(*
SPDX-FileCopyrightText: © 2026 Oleksandr Tiutyk <trofimich@gmail.com>
SPDX-License-Identifier: MIT
License: https://opensource.org/license/mit
*)

(*!
<summary>Enumerates a borrowed collection using an independent cursor.</summary>
<description>
The source must be non-null, outlive the cursor and remain structurally unchanged during traversal. The caller
explicitly releases a dynamically created cursor. Current borrows a byte cached in this cursor, not the source
buffer; it never transfers ownership. MoveNext stops advancing at the end position of an unchanged source;
repeated exhausted calls return FALSE until Reset.
A null constructor source is diagnosed by traversal/current access, never by FB_init.
</description>
*)

{attribute 'no_explicit_call' := 'do not call this function block directly'}
{attribute 'enable_dynamic_creation'}
FUNCTION_BLOCK ByteListEnumerator EXTENDS TOF_Core.Object IMPLEMENTS TOF_Core.IEnumerator
VAR_STAT
	//! <summary>Class name shared by all instances of this function block.</summary>
	{attribute 'hide'} 
	_ClassName : STRING := __POUNAME();
END_VAR
VAR
	{attribute 'hide'} 
	_List : IReadOnlyByteList;
	{attribute 'hide'} 
	_CurrentIndex : DINT := -1;
	
	{attribute 'hide'} 
	_CurrentByte : BYTE;
	{attribute 'hide'} 
	_GenericValue : TOF_Core.GENERIC_VALUE;	
END_VAR

(*!
<summary>Borrows the concrete cursor class name without transferring storage ownership.</summary>
*)
{attribute 'monitoring' := 'call'}
PROPERTY ClassName : REFERENCE TO STRING
GET
ClassName REF= _ClassName;
END_GET
END_PROPERTY

(*!
<summary>Exposes a read-only borrowed view of the current entry.</summary>
<description>
Reading Current before the first successful MoveNext, after Reset or after exhaustion yields an empty
descriptor. At a valid position, the source byte is copied into cursor-local storage and the returned
descriptor borrows that storage, including when the byte value is zero. Do not modify or release the
descriptor. Keep the cursor alive while using the view; subsequent Current access can overwrite its cached
byte. Cursor movement or reset invalidates the previous view contract.
Missing source raises DataMemberNotSpecifiedException before source access or cursor advancement.
</description>
*)
{attribute 'monitoring' := 'call'}
PROPERTY FINAL Current : REFERENCE TO TOF_Core.GENERIC_VALUE
GET
requireSource();

IF _CurrentIndex >= 0 AND_THEN _CurrentIndex < _List.Length THEN
	_CurrentByte := _List.Get(index := _CurrentIndex); 
	_GenericValue := TOF_Core.GenericValueFactory.FromParts(
		genericTypeClass := TOF_Core.GENERIC_TYPE_CLASS.UINT_8,
		address := ADR(_CurrentByte),
		size := 1,
		memoryManagementBehavior := TOF_Core.GENERIC_MEMORY_MANAGEMENT_BEHAVIOR.STORE_ORIGINAL_REFERENCE_AND_NOT_OWNS_MEMORY
	);
ELSE
	_GenericValue.Reset();
END_IF 

Current REF= _GenericValue;
END_GET
END_PROPERTY

(*!
<summary>Returns the current entry in its concrete representation.</summary>
<description>
Use only after MoveNext returns TRUE and before the next cursor or source change. No result is promised
outside a valid position. The byte is returned by value.
Missing source raises DataMemberNotSpecifiedException before source access or cursor advancement.
</description>
*)
{attribute 'monitoring' := 'call'}
PROPERTY FINAL CurrentByte : BYTE
GET
requireSource();

IF _CurrentIndex >= 0 AND_THEN _CurrentIndex < _List.Length THEN
	CurrentByte := _List.Get(index := _CurrentIndex); 
END_IF
END_GET
END_PROPERTY

(*!
<summary>Binds the borrowed source for enumeration.</summary>
<description>
The source must be non-null and outlive the cursor. Only the reference is assigned; no allocation, callbacks
or throwing validation are performed. A null source remains invalid configuration and is reported by
MoveNext or current-value access without throwing from initialization.
</description>
*)
METHOD FB_init : BOOL
VAR_INPUT
	bInitRetains : BOOL; // TRUE: the retain variables are initialized (reset warm / reset cold)
	bInCopyCode : BOOL;  // TRUE: the instance will be copied to the copy code afterward (online change)
	list : IReadOnlyByteList;
END_VAR
_List := list;
END_METHOD

(*!
<summary>Advances the cursor to the next source position.</summary>
<description>
The source must be live, non-null and structurally unchanged during traversal. TRUE identifies a current
entry. The index advances only while below source Length and stops at the end position. Repeated exhausted
calls return FALSE without incrementing the index; reading Current yields an empty descriptor. Reset allows
traversal from the beginning again. No snapshot or mutation detection is provided. Descendants cannot override
this cursor operation; advancement, reset and borrowed current views use the same cursor state.
Missing source raises DataMemberNotSpecifiedException before source access or cursor advancement.
</description>
*)
{attribute "object_name" := "MoveNext"}
METHOD FINAL MoveNext : BOOL
requireSource();

IF _CurrentIndex < _List.Length THEN
	_CurrentIndex := _CurrentIndex + 1;
END_IF

MoveNext := _CurrentIndex < _List.Length;
END_METHOD

(*!
<summary>Provides the library namespace for diagnostics.</summary>
<description>
Borrowed read-only reference to compiler-initialized metadata; no ownership transfer.
</description>
*)
{attribute 'monitoring' := 'call'}
PROPERTY NamespaceName : REFERENCE TO STRING
GET
NamespaceName REF= CurrentNamespace.Name;
END_GET
END_PROPERTY

(*!
<summary>Places the cursor before the first source entry.</summary>
<description>
The next MoveNext starts at zero. Does not modify the source or release payload; reading Current now yields an
empty descriptor. Descendants cannot override this cursor operation; advancement, reset and borrowed current
views use the same cursor state.
</description>
*)
{attribute "object_name" := "Reset"}
METHOD FINAL Reset
_CurrentIndex := -1;
END_METHOD

(*!
<summary>Reports the size of this function-block instance.</summary>
<description>
Measured in bytes; includes inline storage but excludes separately allocated buffers, payload and enumerators.
</description>
*)
{attribute 'monitoring' := 'call'}
PROPERTY SelfSize : ULINT
GET
SelfSize := XSIZEOF(THIS^);
END_GET
END_PROPERTY

(*!
<summary>Requires the configured source before traversal or current-value access.</summary>
<description>
A missing mandatory source is configuration failure, not an empty collection. Raises a framework diagnostic
outside lifecycle methods and before mutation; it does not validate arbitrary pointer lifetime.
</description>
*)
METHOD PRIVATE requireSource
IF _List = 0 THEN
	TOF_Core.Exceptions.ThrowDataMemberNotSpecified(
		sourceNamespaceName := NamespaceName,
		sourceClassName := ClassName,
		sourcePOUName := __POUNAME(),
		sourcePosition := __POSITION(),
		dataMemberName := 'list'
	);
END_IF
END_METHOD

END_FUNCTION_BLOCK

(* stored: Version 1.1.0.1
   POU ByteListEnumerator: Id {0eaa5e30-f578-440b-bf42-b39d6e892a5e}, SpecialFunc None
   Property ClassName: Id {d0ef8e8d-8cab-4592-a439-a079fcf6b703}
   Get Get: Id {0311af57-34ad-4839-8f64-45605666dbff}
   Property Current: Id {34633660-6766-4502-8d0b-2f6866bc7750}
   Get Get: Id {a7991f02-dccd-4bc0-a616-ec473de5b639}
   Property CurrentByte: Id {110179b3-6f98-4cf4-ae85-eec25b6472ac}
   Get Get: Id {15812a15-c7f7-49c5-8a38-6b883ff80d77}
   Method FB_init: Id {64a9e57e-1291-4061-b0c2-def30792e0f4}
   Method MoveNext: Id {bb301441-6417-4b6a-8920-265d238eecbf}
   Property NamespaceName: Id {3f49bd54-cf7c-48ab-b476-040534a96221}
   Get Get: Id {04eab4d1-eee5-42eb-828c-34eca7f6264d}
   Method Reset: Id {1a671f16-85bb-4034-972d-cf14ae393e20}
   Property SelfSize: Id {108df5a2-3a30-4039-b541-048811bab97b}
   Get Get: Id {de7624c7-c9a3-4045-8ace-16907f6279e5}
   Method requireSource: Id {1464e6f8-e464-4557-a4d3-0cf8e2184a1a} *)
